(* Logix 5000 project; controller Uidaho_Factory vendor 1 type 14 code 165 rev 38.11; software revision 38.00; part 3 of 3 *)
(* tags used below, declared in another part *)
   MPO_Done : BOOL;
   MPO_Turntable_Start : BOOL;
   SLD_Blue_Min : DINT;
   SLD_Blue_Time : DINT;
   SLD_Min_Value : DINT;
   SLD_Move_Time : DINT;
   SLD_Normal : DINT;
   SLD_Red_Min : DINT;
   SLD_Red_Time : DINT;
   SLD_start : DINT;
   SLD_Step : DINT;
   SLD_White_Time : DINT;
   Step : DINT[20];
   StepTimers : TIMER[20];
   TurntableTimers : TIMER[10];
   PWM_Outputs : PWM_Out[20];
   Scaled_Analog_Color_Sensor_SLD : DINT;   // SLD - A1 = Color sensor
(* MainProgram, continued *)

ROUTINE MPO_Turntable_Process   (* ladder *)
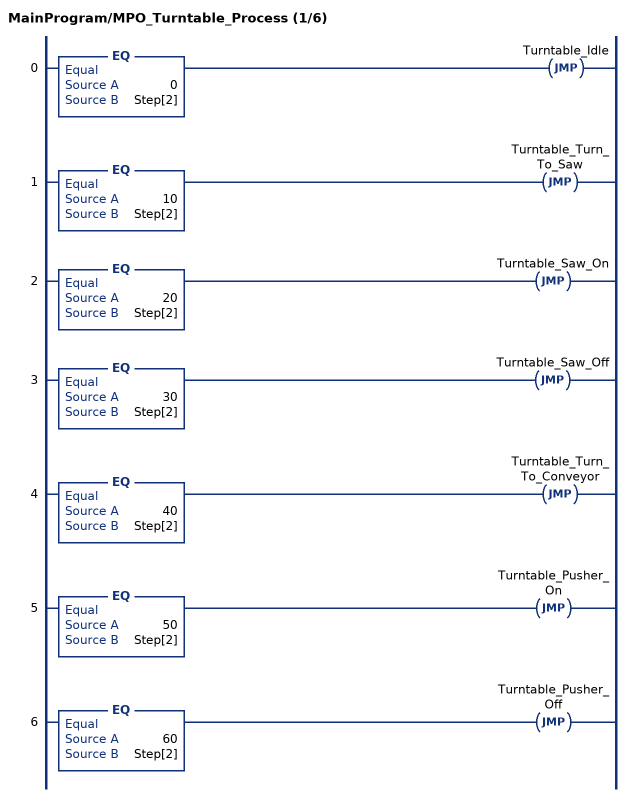
   0: EQ(0,Step[2])JMP(Turntable_Idle);
   1: EQ(10,Step[2])JMP(Turntable_Turn_To_Saw);
   2: EQ(20,Step[2])JMP(Turntable_Saw_On);
   3: EQ(30,Step[2])JMP(Turntable_Saw_Off);
   4: EQ(40,Step[2])JMP(Turntable_Turn_To_Conveyor);
   5: EQ(50,Step[2])JMP(Turntable_Pusher_On);
   6: EQ(60,Step[2])JMP(Turntable_Pusher_Off);
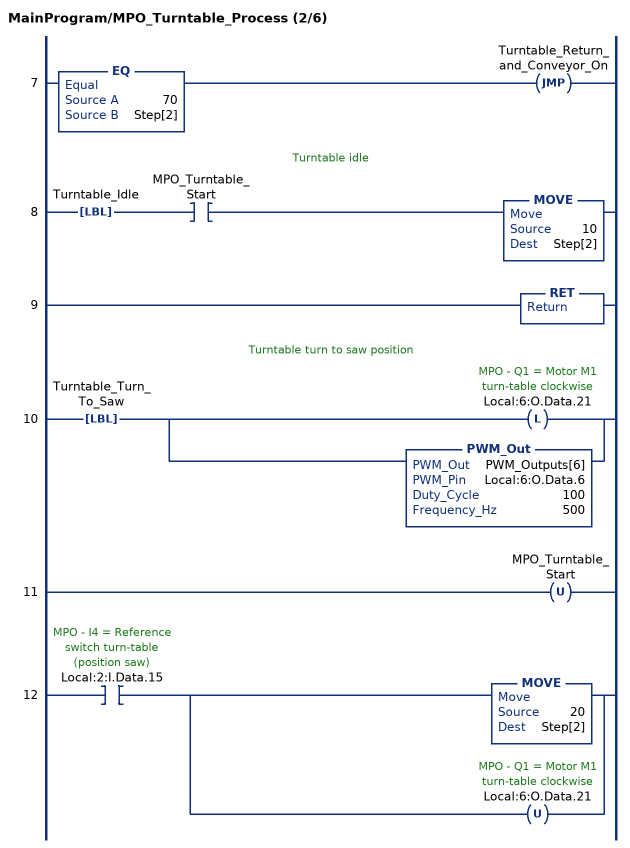
   7: EQ(70,Step[2])JMP(Turntable_Return_and_Conveyor_On);
   // Turntable idle
   8: LBL(Turntable_Idle)XIC(MPO_Turntable_Start)MOVE(10,Step[2]);
   9: RET();
   // Turntable turn to saw position
   10: LBL(Turntable_Turn_To_Saw)[OTL(Local:6:O.Data.21) ,PWM_Out(PWM_Outputs[6],Local:6:O.Data.6,100,500) ];
   11: OTU(MPO_Turntable_Start);
   12: XIC(Local:2:I.Data.15)[MOVE(20,Step[2]) ,OTU(Local:6:O.Data.21) ];
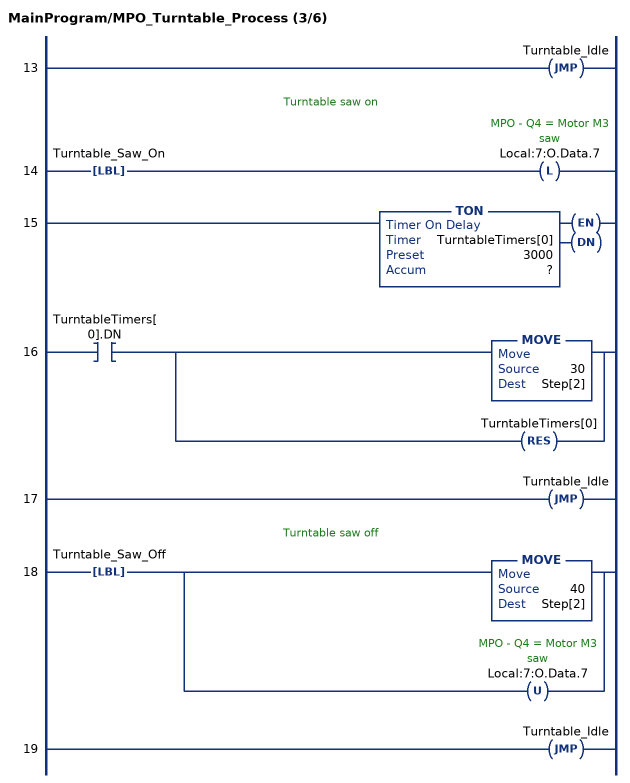
   13: JMP(Turntable_Idle);
   // Turntable saw on
   14: LBL(Turntable_Saw_On)OTL(Local:7:O.Data.7);
   15: TON(TurntableTimers[0],?,?);
   16: XIC(TurntableTimers[0].DN)[MOVE(30,Step[2]) ,RES(TurntableTimers[0]) ];
   17: JMP(Turntable_Idle);
   // Turntable saw off
   18: LBL(Turntable_Saw_Off)[MOVE(40,Step[2]) ,OTU(Local:7:O.Data.7) ];
   19: JMP(Turntable_Idle);
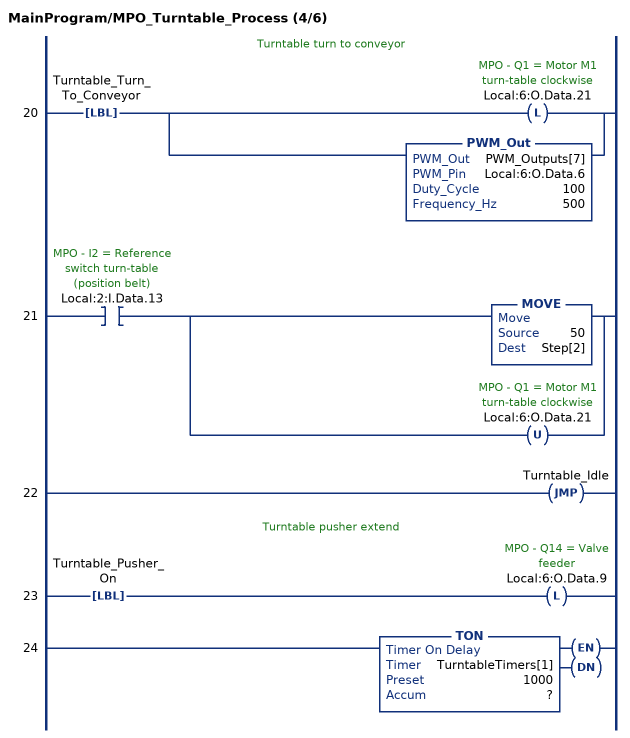
   // Turntable turn to conveyor
   20: LBL(Turntable_Turn_To_Conveyor)[OTL(Local:6:O.Data.21) ,PWM_Out(PWM_Outputs[7],Local:6:O.Data.6,100,500) ];
   21: XIC(Local:2:I.Data.13)[MOVE(50,Step[2]) ,OTU(Local:6:O.Data.21) ];
   22: JMP(Turntable_Idle);
   // Turntable pusher extend
   23: LBL(Turntable_Pusher_On)OTL(Local:6:O.Data.9);
   24: TON(TurntableTimers[1],?,?);
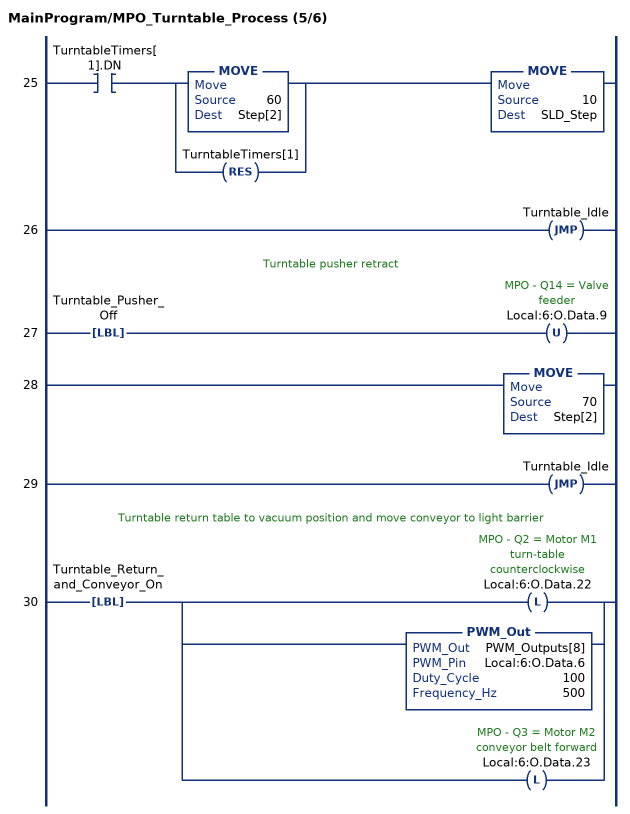
   25: XIC(TurntableTimers[1].DN)[MOVE(60,Step[2]) ,RES(TurntableTimers[1]) ]MOVE(10,SLD_Step);
   26: JMP(Turntable_Idle);
   // Turntable pusher retract
   27: LBL(Turntable_Pusher_Off)OTU(Local:6:O.Data.9);
   28: MOVE(70,Step[2]);
   29: JMP(Turntable_Idle);
   // Turntable return table to vacuum position and move conveyor to light barrier
   30: LBL(Turntable_Return_and_Conveyor_On)[[OTL(Local:6:O.Data.22) ,PWM_Out(PWM_Outputs[8],Local:6:O.Data.6,100,500) ] ,OTL(Local:6:O.Data.23) ];
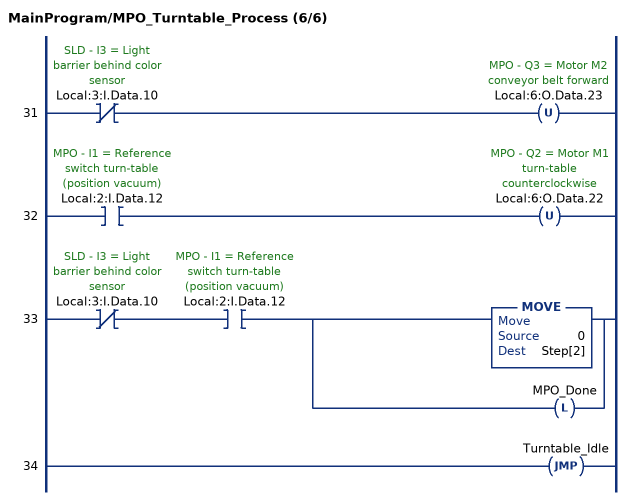
   31: XIO(Local:3:I.Data.10)OTU(Local:6:O.Data.23);
   32: XIC(Local:2:I.Data.12)OTU(Local:6:O.Data.22);
   33: XIO(Local:3:I.Data.10)XIC(Local:2:I.Data.12)[MOVE(0,Step[2]) ,OTL(MPO_Done) ];
   34: JMP(Turntable_Idle);
END_ROUTINE

ROUTINE SLD_Controller   (* ladder *)
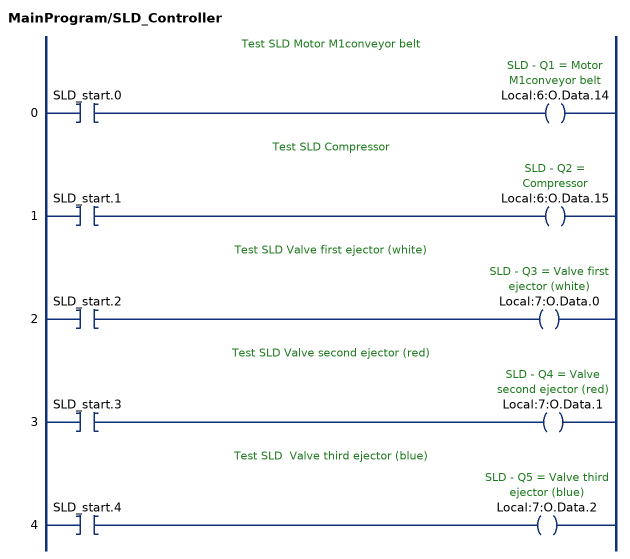
   // Test SLD Motor M1conveyor belt
   0: XIC(SLD_start.0)OTE(Local:6:O.Data.14);
   // Test SLD Compressor
   1: XIC(SLD_start.1)OTE(Local:6:O.Data.15);
   // Test SLD Valve first ejector (white)
   2: XIC(SLD_start.2)OTE(Local:7:O.Data.0);
   // Test SLD Valve second ejector (red)
   3: XIC(SLD_start.3)OTE(Local:7:O.Data.1);
   // Test SLD  Valve third ejector (blue)
   4: XIC(SLD_start.4)OTE(Local:7:O.Data.2);
END_ROUTINE

ROUTINE SLD_Sequencer   (* ladder *)
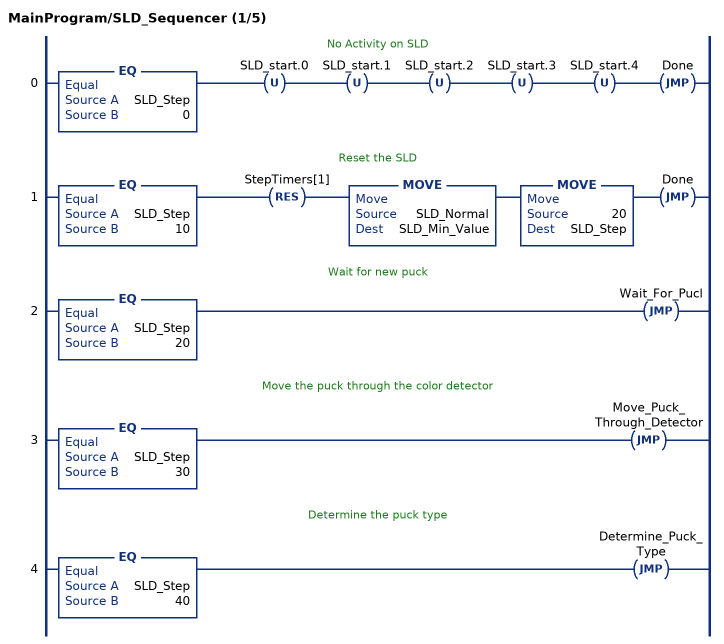
   // No Activity on SLD
   0: EQ(SLD_Step,0)OTU(SLD_start.0)OTU(SLD_start.1)OTU(SLD_start.2)OTU(SLD_start.3)OTU(SLD_start.4)JMP(Done);
   // Reset the SLD
   1: EQ(SLD_Step,10)RES(StepTimers[1])MOVE(SLD_Normal,SLD_Min_Value)MOVE(20,SLD_Step)JMP(Done);
   // Wait for new puck
   2: EQ(SLD_Step,20)JMP(Wait_For_Pucl);
   // Move the puck through the color detector
   3: EQ(SLD_Step,30)JMP(Move_Puck_Through_Detector);
   // Determine the puck type
   4: EQ(SLD_Step,40)JMP(Determine_Puck_Type);
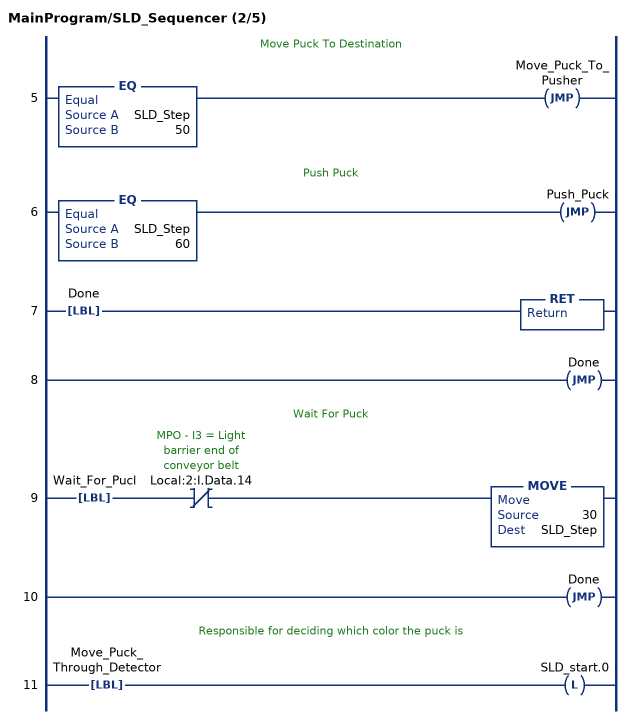
   // Move Puck To Destination
   5: EQ(SLD_Step,50)JMP(Move_Puck_To_Pusher);
   // Push Puck
   6: EQ(SLD_Step,60)JMP(Push_Puck);
   7: LBL(Done)RET();
   8: JMP(Done);
   // Wait For Puck
   9: LBL(Wait_For_Pucl)XIO(Local:2:I.Data.14)MOVE(30,SLD_Step);
   10: JMP(Done);
   // Responsible for deciding which color the puck is
   11: LBL(Move_Puck_Through_Detector)OTL(SLD_start.0);
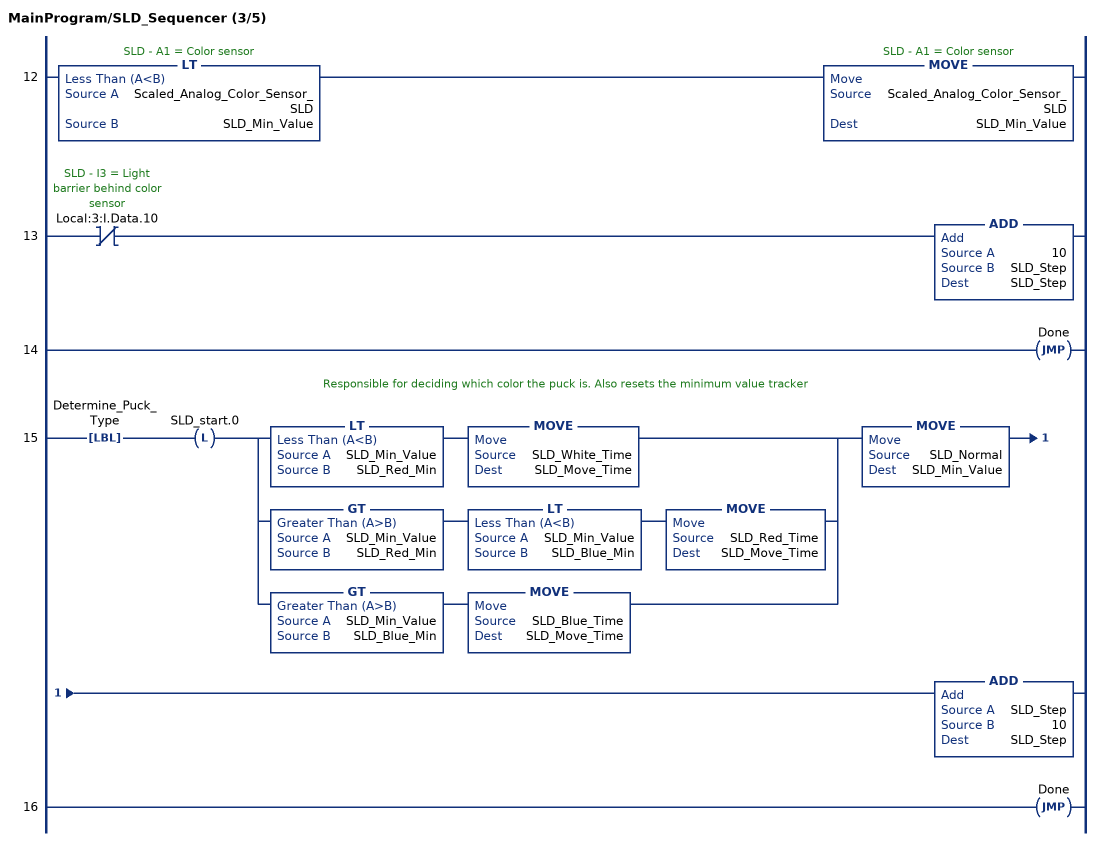
   12: LT(Scaled_Analog_Color_Sensor_SLD,SLD_Min_Value)MOVE(Scaled_Analog_Color_Sensor_SLD,SLD_Min_Value);
   13: XIO(Local:3:I.Data.10)ADD(10,SLD_Step,SLD_Step);
   14: JMP(Done);
   // Responsible for deciding which color the puck is. Also resets the minimum value tracker
   15: LBL(Determine_Puck_Type)OTL(SLD_start.0)[LT(SLD_Min_Value,SLD_Red_Min) MOVE(SLD_White_Time,SLD_Move_Time) ,GT(SLD_Min_Value,SLD_Red_Min) LT(SLD_Min_Value,SLD_Blue_Min) MOVE(SLD_Red_Time,SLD_Move_Time) ,GT(SLD_Min_Value,SLD_Blue_Min) MOVE(SLD_Blue_Time,SLD_Move_Time) ]MOVE(SLD_Normal,SLD_Min_Value)ADD(SLD_Step,10,SLD_Step);
   16: JMP(Done);
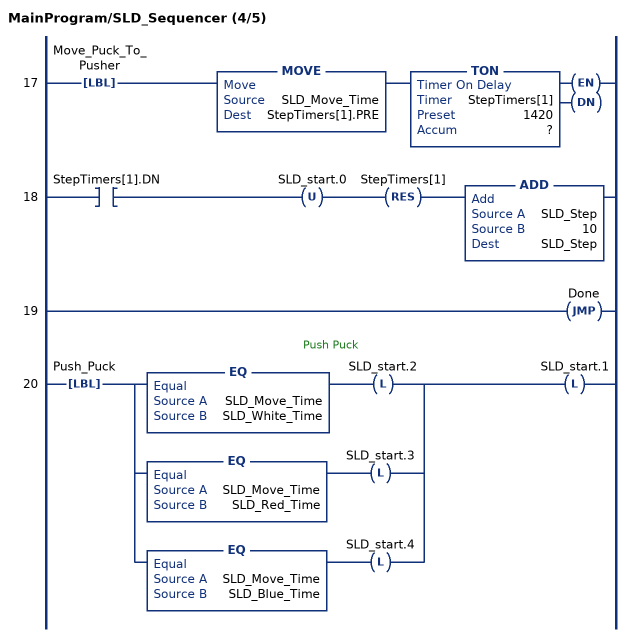
   17: LBL(Move_Puck_To_Pusher)MOVE(SLD_Move_Time,StepTimers[1].PRE)TON(StepTimers[1],?,?);
   18: XIC(StepTimers[1].DN)OTU(SLD_start.0)RES(StepTimers[1])ADD(SLD_Step,10,SLD_Step);
   19: JMP(Done);
   // Push Puck
   20: LBL(Push_Puck)[EQ(SLD_Move_Time,SLD_White_Time) OTL(SLD_start.2) ,EQ(SLD_Move_Time,SLD_Red_Time) OTL(SLD_start.3) ,EQ(SLD_Move_Time,SLD_Blue_Time) OTL(SLD_start.4) ]OTL(SLD_start.1);
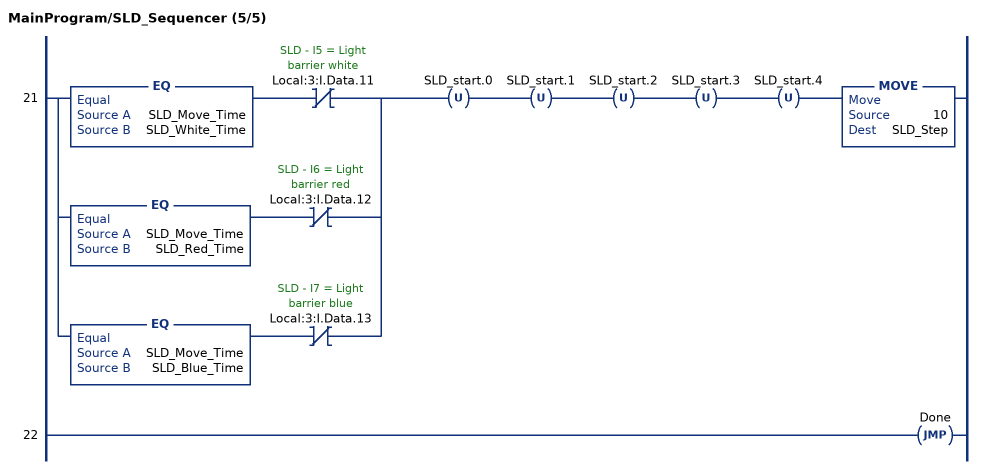
   21: [EQ(SLD_Move_Time,SLD_White_Time) XIO(Local:3:I.Data.11) ,EQ(SLD_Move_Time,SLD_Red_Time) XIO(Local:3:I.Data.12) ,EQ(SLD_Move_Time,SLD_Blue_Time) XIO(Local:3:I.Data.13) ]OTU(SLD_start.0)OTU(SLD_start.1)OTU(SLD_start.2)OTU(SLD_start.3)OTU(SLD_start.4)MOVE(10,SLD_Step);
   22: JMP(Done);
END_ROUTINE
END_PROGRAM
